TYPE ST_SVs_504_505_Zustand :
STRUCT
	Stellung_Anford				: BOOL;
	Stellung_Soll				: BOOL;
	Stellung					: BOOL;

	Stellungrueckmeldung0_504	: BOOL;
	Stellungrueckmeldung1_504	: BOOL;

	Stellungrueckmeldung0_505	: BOOL;
	Stellungrueckmeldung1_505	: BOOL;

	Freigabe					: BOOL;
	Freigabe_Deakt				: BOOL;
	Freigabe_Code				: WORD;

	Stoerung					: BOOL;
	Stoerung_Code				: WORD;

	Warnung						: BOOL;
	Warnung_Code				: WORD;

	Status						: SINT;

	Stellungwechsel01			: BOOL;
	Stellungwechsel10			: BOOL;

	Quittierung					: BOOL;

END_STRUCT
END_TYPE

(* stored: Version 1.1.0.1, ProductVersion 3.1.4024.9
   DUT ST_SVs_504_505_Zustand: Id {e6854c62-c000-4b8d-9e69-3303dbc350f9} *)
